SUBAPPLICATION Klappen (* Subapplication Type *)
  (* Standard: 61499-2 *)
  (* Version 1.0, 2023-01-29, Franz *)
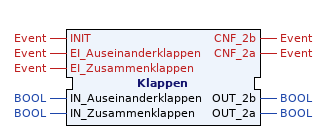
  EVENT_INPUT
    INIT;
    EI_Auseinanderklappen;
    EI_Zusammenklappen;
  END_EVENT
  EVENT_OUTPUT
    CNF_2b;
    CNF_2a;
  END_EVENT
  VAR_INPUT
    IN_Auseinanderklappen : BOOL;
    IN_Zusammenklappen : BOOL;
  END_VAR
  VAR_OUTPUT
    OUT_2b : BOOL;
    OUT_2a : BOOL;
  END_VAR
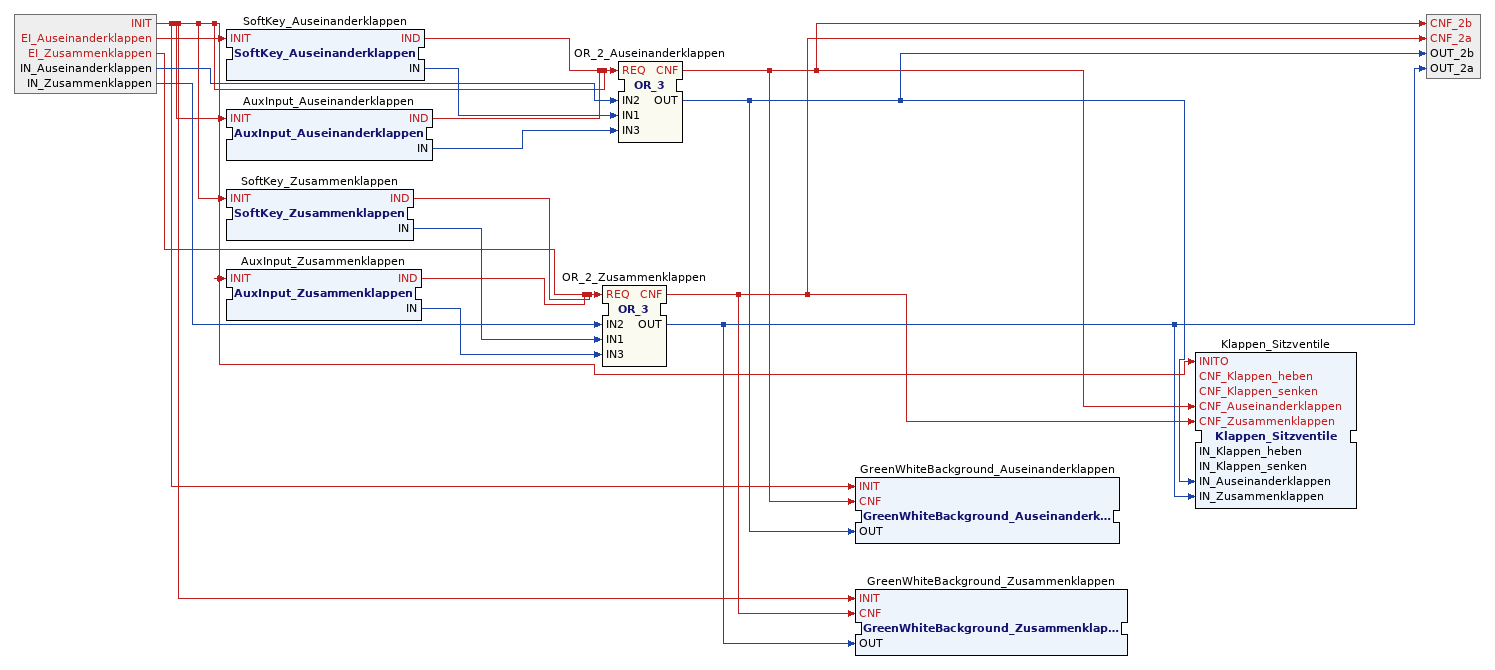
  FBS
    OR_2_Auseinanderklappen : OR_3;
    OR_2_Zusammenklappen : OR_3;
  END_FBS
  SUBAPPS
    GreenWhiteBackground_Auseinanderklappen : GreenWhiteBackground_Auseinanderklappen;
    GreenWhiteBackground_Zusammenklappen : GreenWhiteBackground_Zusammenklappen;
    Klappen_Sitzventile : Klappen_Sitzventile;
    SoftKey_Auseinanderklappen : SoftKey_Auseinanderklappen;
    SoftKey_Zusammenklappen : SoftKey_Zusammenklappen;
    AuxInput_Zusammenklappen : AuxInput_Zusammenklappen;
    AuxInput_Auseinanderklappen : AuxInput_Auseinanderklappen;
  END_SUBAPPS
  EVENT_CONNECTIONS
    INIT TO GreenWhiteBackground_Auseinanderklappen.INIT;
    INIT TO GreenWhiteBackground_Zusammenklappen.INIT;
    INIT TO Klappen_Sitzventile.INITO;
    EI_Auseinanderklappen TO OR_2_Auseinanderklappen.REQ;
    OR_2_Auseinanderklappen.CNF TO GreenWhiteBackground_Auseinanderklappen.CNF;
    OR_2_Auseinanderklappen.CNF TO Klappen_Sitzventile.CNF_Auseinanderklappen;
    EI_Zusammenklappen TO OR_2_Zusammenklappen.REQ;
    OR_2_Zusammenklappen.CNF TO GreenWhiteBackground_Zusammenklappen.CNF;
    OR_2_Zusammenklappen.CNF TO Klappen_Sitzventile.CNF_Zusammenklappen;
    INIT TO SoftKey_Auseinanderklappen.INIT;
    SoftKey_Auseinanderklappen.IND TO OR_2_Auseinanderklappen.REQ;
    INIT TO SoftKey_Zusammenklappen.INIT;
    SoftKey_Zusammenklappen.IND TO OR_2_Zusammenklappen.REQ;
    INIT TO AuxInput_Zusammenklappen.INIT;
    AuxInput_Zusammenklappen.IND TO OR_2_Zusammenklappen.REQ;
    INIT TO AuxInput_Auseinanderklappen.INIT;
    AuxInput_Auseinanderklappen.IND TO OR_2_Auseinanderklappen.REQ;
    OR_2_Auseinanderklappen.CNF TO CNF_2b;
    OR_2_Zusammenklappen.CNF TO CNF_2a;
  END_CONNECTIONS
  DATA_CONNECTIONS
    IN_Auseinanderklappen TO OR_2_Auseinanderklappen.IN2;
    OR_2_Auseinanderklappen.OUT TO GreenWhiteBackground_Auseinanderklappen.OUT;
    OR_2_Auseinanderklappen.OUT TO Klappen_Sitzventile.IN_Auseinanderklappen;
    IN_Zusammenklappen TO OR_2_Zusammenklappen.IN2;
    OR_2_Zusammenklappen.OUT TO GreenWhiteBackground_Zusammenklappen.OUT;
    OR_2_Zusammenklappen.OUT TO Klappen_Sitzventile.IN_Zusammenklappen;
    SoftKey_Auseinanderklappen.IN TO OR_2_Auseinanderklappen.IN1;
    SoftKey_Zusammenklappen.IN TO OR_2_Zusammenklappen.IN1;
    AuxInput_Zusammenklappen.IN TO OR_2_Zusammenklappen.IN3;
    AuxInput_Auseinanderklappen.IN TO OR_2_Auseinanderklappen.IN3;
    OR_2_Auseinanderklappen.OUT TO OUT_2b;
    OR_2_Zusammenklappen.OUT TO OUT_2a;
  END_CONNECTIONS
END_SUBAPPLICATION
